INTERFACE I_Command

METHOD Execute
VAR_INPUT
END_VAR
END_METHOD

END_INTERFACE

(* stored: Version 1.1.0.1, ProductVersion 3.1.4024.5
   Itf I_Command: Id {28050084-7919-40a7-8c66-8b1649566e1f}
   Method Execute: Id {25629016-2c43-40ba-8923-5d275b229e74} *)
